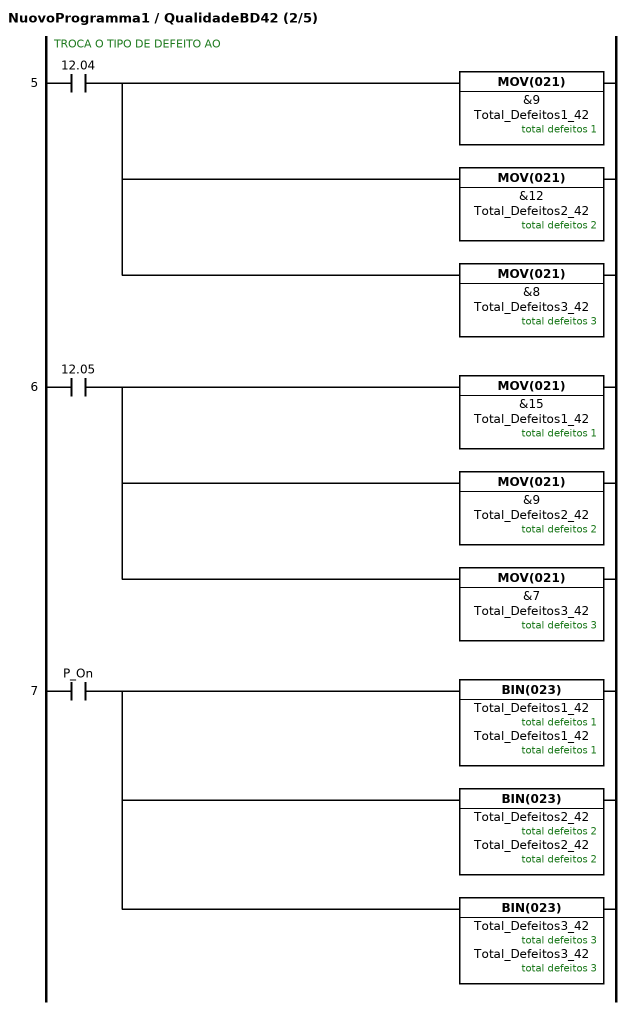
; [picture p24: NuovoProgramma1 / QualidadeBD42, rungs 5-7]
; rung 5: TROCA O TIPO DE DEFEITO AO
LD 12.04
MOV(021) &9 Total_Defeitos1_42  ; total defeitos 1
MOV(021) &12 Total_Defeitos2_42  ; total defeitos 2
MOV(021) &8 Total_Defeitos3_42  ; total defeitos 3
; rung 6
LD 12.05
MOV(021) &15 Total_Defeitos1_42  ; total defeitos 1
MOV(021) &9 Total_Defeitos2_42  ; total defeitos 2
MOV(021) &7 Total_Defeitos3_42  ; total defeitos 3
; rung 7
LD P_On
BIN(023) Total_Defeitos1_42 Total_Defeitos1_42  ; total defeitos 1
BIN(023) Total_Defeitos2_42 Total_Defeitos2_42  ; total defeitos 2
BIN(023) Total_Defeitos3_42 Total_Defeitos3_42  ; total defeitos 3

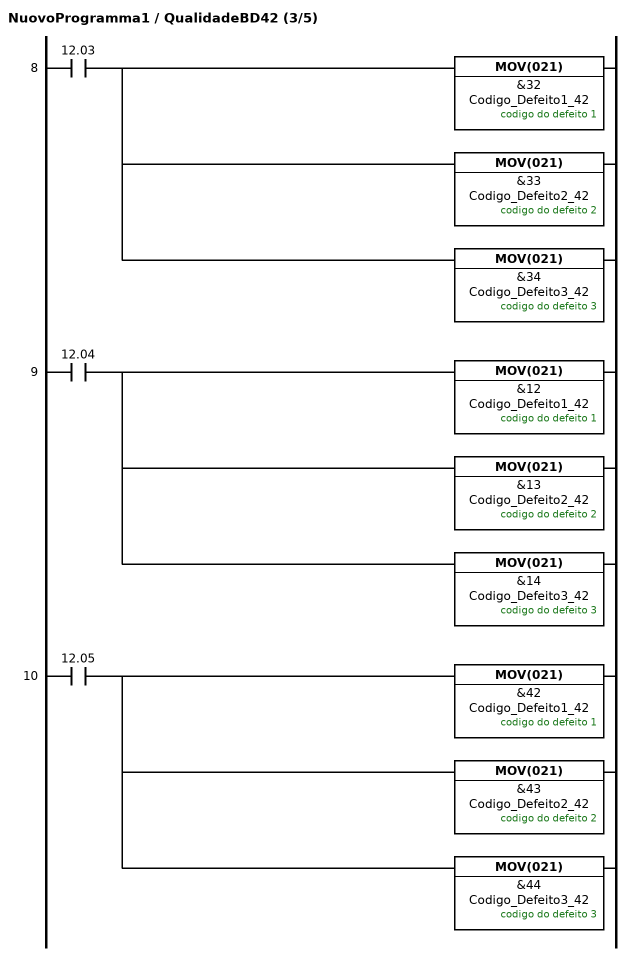
; rung 8
LD 12.03
MOV(021) &32 Codigo_Defeito1_42  ; codigo do defeito 1
MOV(021) &33 Codigo_Defeito2_42  ; codigo do defeito 2
MOV(021) &34 Codigo_Defeito3_42  ; codigo do defeito 3
; rung 9
LD 12.04
MOV(021) &12 Codigo_Defeito1_42  ; codigo do defeito 1
MOV(021) &13 Codigo_Defeito2_42  ; codigo do defeito 2
MOV(021) &14 Codigo_Defeito3_42  ; codigo do defeito 3
; rung 10
LD 12.05
MOV(021) &42 Codigo_Defeito1_42  ; codigo do defeito 1
MOV(021) &43 Codigo_Defeito2_42  ; codigo do defeito 2
MOV(021) &44 Codigo_Defeito3_42  ; codigo do defeito 3

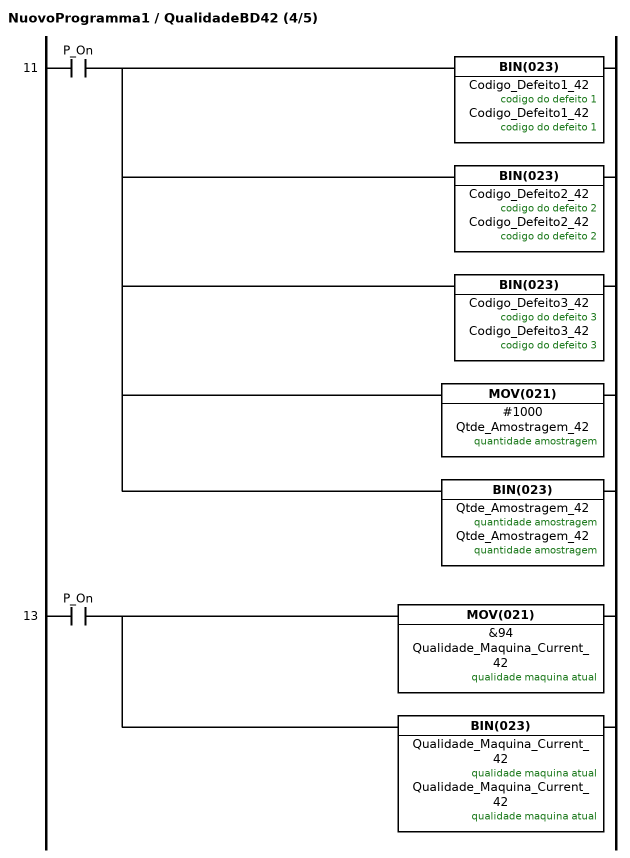
; rung 11
LD P_On
BIN(023) Codigo_Defeito1_42 Codigo_Defeito1_42  ; codigo do defeito 1
BIN(023) Codigo_Defeito2_42 Codigo_Defeito2_42  ; codigo do defeito 2
BIN(023) Codigo_Defeito3_42 Codigo_Defeito3_42  ; codigo do defeito 3
MOV(021) #1000 Qtde_Amostragem_42  ; quantidade amostragem
BIN(023) Qtde_Amostragem_42 Qtde_Amostragem_42  ; quantidade amostragem
; rung 13
LD P_On
MOV(021) &94 Qualidade_Maquina_Current_42  ; qualidade maquina atual
BIN(023) Qualidade_Maquina_Current_42 Qualidade_Maquina_Current_42  ; qualidade maquina atual

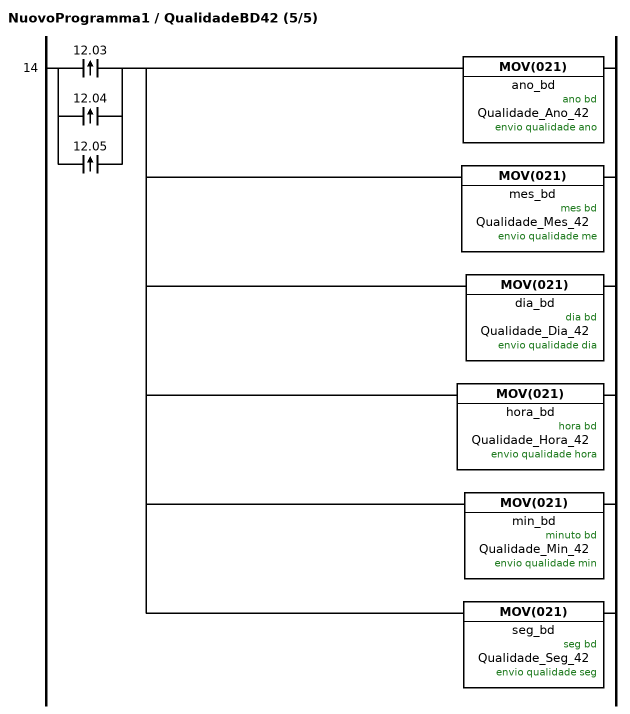
; rung 14
@LD 12.03
@OR 12.04
@OR 12.05
MOV(021) ano_bd Qualidade_Ano_42  ; ano bd, envio qualidade ano
MOV(021) mes_bd Qualidade_Mes_42  ; mes bd, envio qualidade me
MOV(021) dia_bd Qualidade_Dia_42  ; dia bd, envio qualidade dia
MOV(021) hora_bd Qualidade_Hora_42  ; hora bd, envio qualidade hora
MOV(021) min_bd Qualidade_Min_42  ; minuto bd, envio qualidade min
MOV(021) seg_bd Qualidade_Seg_42  ; seg bd, envio qualidade seg

### Section QualidadeBD43

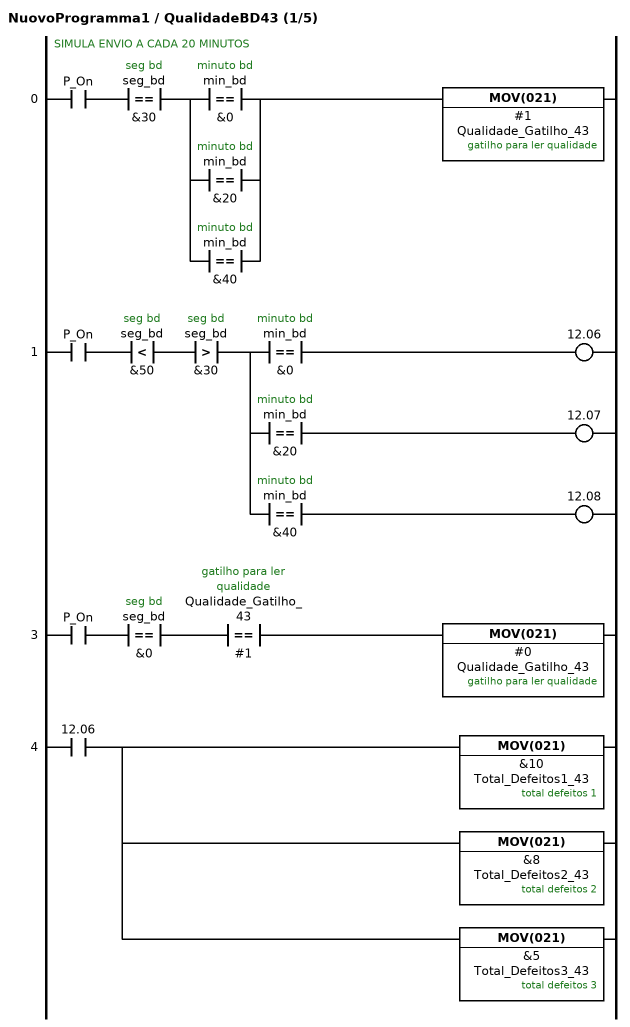
; rung 0: SIMULA ENVIO A CADA 20 MINUTOS
LD P_On
AND=(300) seg_bd &30  ; seg bd
LD=(300) min_bd &0  ; minuto bd
OR=(300) min_bd &20  ; minuto bd
OR=(300) min_bd &40  ; minuto bd
ANDLD
MOV(021) #1 Qualidade_Gatilho_43  ; gatilho para ler qualidade
; rung 1
LD P_On
AND<(310) seg_bd &50  ; seg bd
AND>(320) seg_bd &30  ; seg bd
OUT TR0
AND=(300) min_bd &0  ; minuto bd
OUT 12.06
LD TR0
AND=(300) min_bd &20  ; minuto bd
OUT 12.07
LD TR0
AND=(300) min_bd &40  ; minuto bd
OUT 12.08
; rung 3
LD P_On
AND=(300) seg_bd &0  ; seg bd
AND=(300) Qualidade_Gatilho_43 #1  ; gatilho para ler qualidade
MOV(021) #0 Qualidade_Gatilho_43  ; gatilho para ler qualidade
; rung 4
LD 12.06
MOV(021) &10 Total_Defeitos1_43  ; total defeitos 1
MOV(021) &8 Total_Defeitos2_43  ; total defeitos 2
MOV(021) &5 Total_Defeitos3_43  ; total defeitos 3

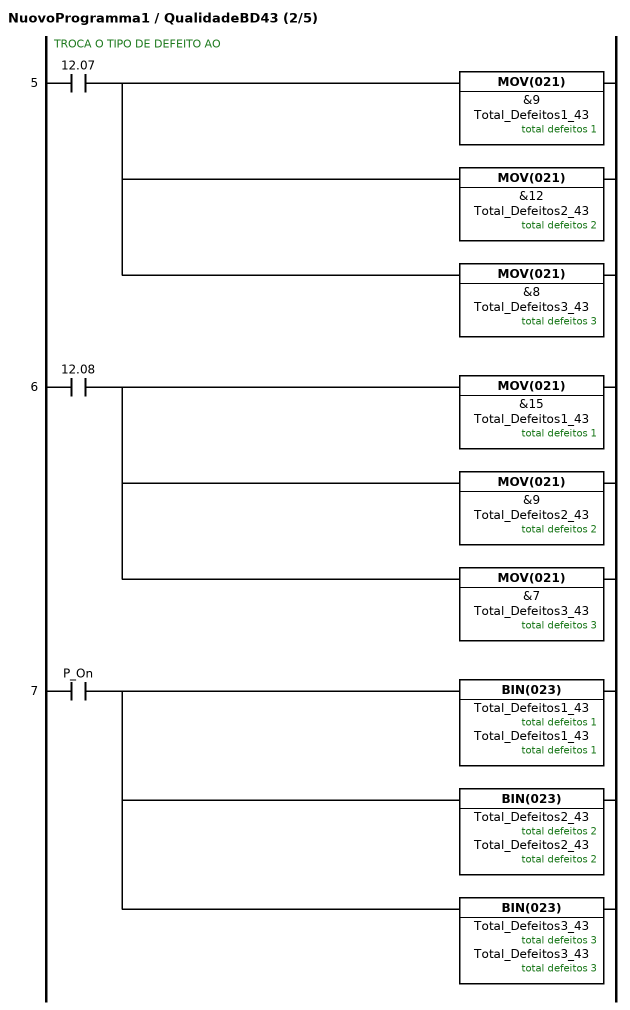
; rung 5: TROCA O TIPO DE DEFEITO AO
LD 12.07
MOV(021) &9 Total_Defeitos1_43  ; total defeitos 1
MOV(021) &12 Total_Defeitos2_43  ; total defeitos 2
MOV(021) &8 Total_Defeitos3_43  ; total defeitos 3
; rung 6
LD 12.08
MOV(021) &15 Total_Defeitos1_43  ; total defeitos 1
MOV(021) &9 Total_Defeitos2_43  ; total defeitos 2
MOV(021) &7 Total_Defeitos3_43  ; total defeitos 3
; rung 7
LD P_On
BIN(023) Total_Defeitos1_43 Total_Defeitos1_43  ; total defeitos 1
BIN(023) Total_Defeitos2_43 Total_Defeitos2_43  ; total defeitos 2
BIN(023) Total_Defeitos3_43 Total_Defeitos3_43  ; total defeitos 3

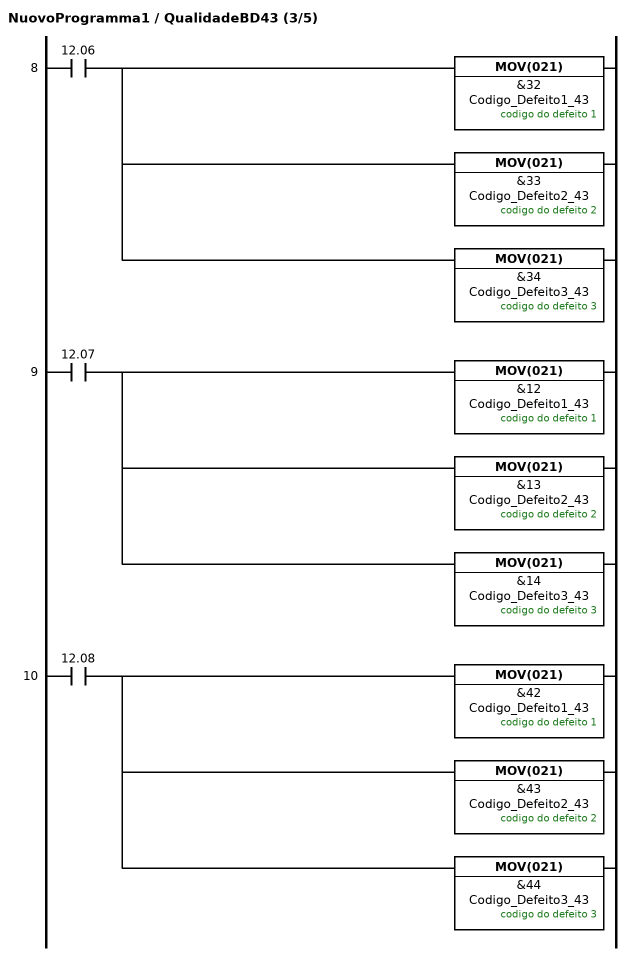
; rung 8
LD 12.06
MOV(021) &32 Codigo_Defeito1_43  ; codigo do defeito 1
MOV(021) &33 Codigo_Defeito2_43  ; codigo do defeito 2
MOV(021) &34 Codigo_Defeito3_43  ; codigo do defeito 3
; rung 9
LD 12.07
MOV(021) &12 Codigo_Defeito1_43  ; codigo do defeito 1
MOV(021) &13 Codigo_Defeito2_43  ; codigo do defeito 2
MOV(021) &14 Codigo_Defeito3_43  ; codigo do defeito 3
; rung 10
LD 12.08
MOV(021) &42 Codigo_Defeito1_43  ; codigo do defeito 1
MOV(021) &43 Codigo_Defeito2_43  ; codigo do defeito 2
MOV(021) &44 Codigo_Defeito3_43  ; codigo do defeito 3

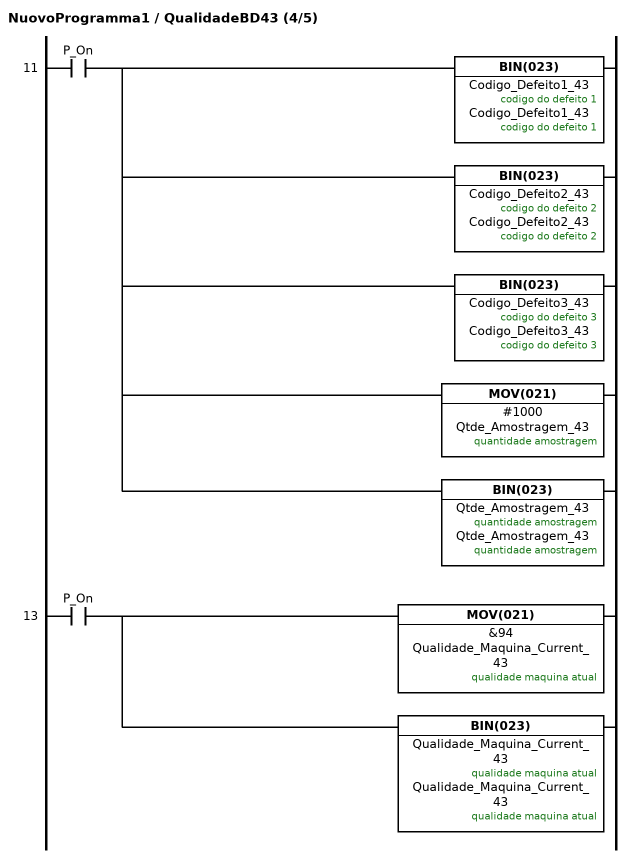
; rung 11
LD P_On
BIN(023) Codigo_Defeito1_43 Codigo_Defeito1_43  ; codigo do defeito 1
BIN(023) Codigo_Defeito2_43 Codigo_Defeito2_43  ; codigo do defeito 2
BIN(023) Codigo_Defeito3_43 Codigo_Defeito3_43  ; codigo do defeito 3
MOV(021) #1000 Qtde_Amostragem_43  ; quantidade amostragem
BIN(023) Qtde_Amostragem_43 Qtde_Amostragem_43  ; quantidade amostragem
; rung 13
LD P_On
MOV(021) &94 Qualidade_Maquina_Current_43  ; qualidade maquina atual
BIN(023) Qualidade_Maquina_Current_43 Qualidade_Maquina_Current_43  ; qualidade maquina atual

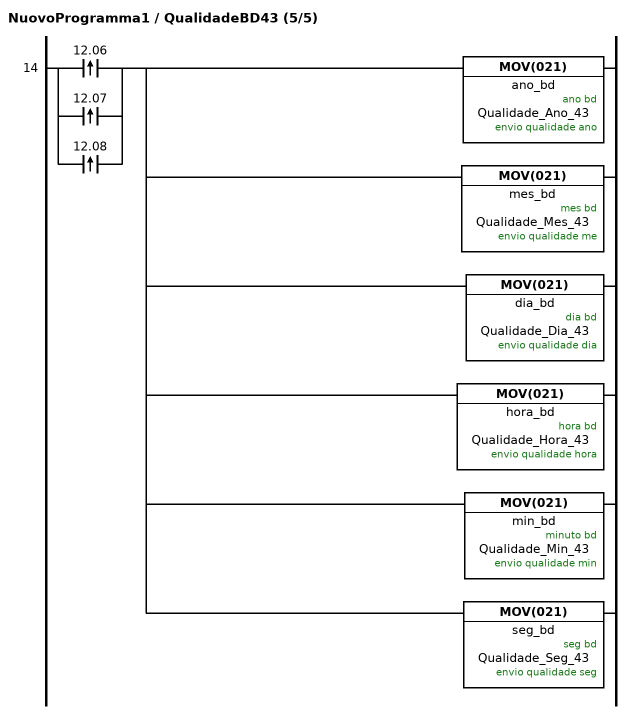
; rung 14
@LD 12.06
@OR 12.07
@OR 12.08
MOV(021) ano_bd Qualidade_Ano_43  ; ano bd, envio qualidade ano
MOV(021) mes_bd Qualidade_Mes_43  ; mes bd, envio qualidade me
MOV(021) dia_bd Qualidade_Dia_43  ; dia bd, envio qualidade dia
MOV(021) hora_bd Qualidade_Hora_43  ; hora bd, envio qualidade hora
MOV(021) min_bd Qualidade_Min_43  ; minuto bd, envio qualidade min
MOV(021) seg_bd Qualidade_Seg_43  ; seg bd, envio qualidade seg

### Section END
; rung 0
END(001)

## Function block Contador_de_Peças_PH29
VAR_INPUT
  Relógio_horas : WORD;
  Relógio_minutos : WORD;
  Dia_calendario : WORD;
  Mês_calendario : WORD;
  Contador : BOOL;
END_VAR
VAR
  _31dias_vezes_2 AT D520 : WORD;
  Ponteiro_DWord AT D522 : WORD;
  Memória_de_Armazenagem AT D524 : WORD;
  Memoria_contagem_BIN AT D526 : WORD;
  Memoria_contagem_BCD AT D528 : WORD;
END_VAR

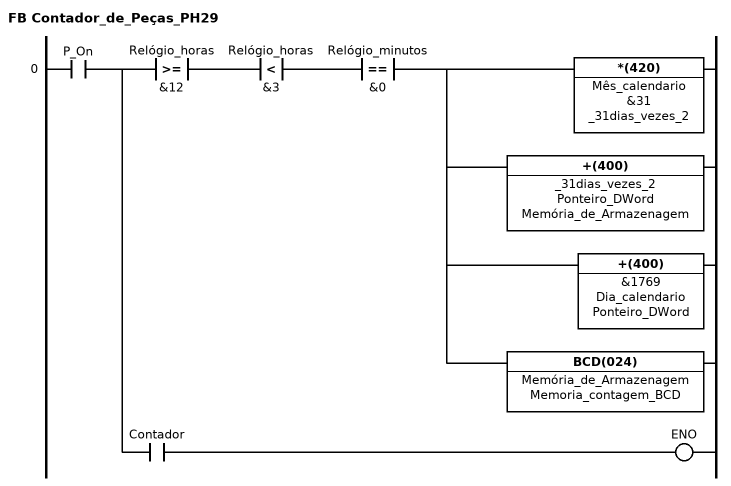
; rung 0
LD P_On
OUT TR0
AND>=(325) Relógio_horas &12
AND<(310) Relógio_horas &3
AND=(300) Relógio_minutos &0
*(420) Mês_calendario &31 _31dias_vezes_2
+(400) _31dias_vezes_2 Ponteiro_DWord Memória_de_Armazenagem
+(400) &1769 Dia_calendario Ponteiro_DWord
BCD(024) Memória_de_Armazenagem Memoria_contagem_BCD
LD TR0
AND Contador
OUT ENO

## Function block Contador_de_Peças_PH30
VAR_INPUT
  Relógio_horas : WORD;
  Relógio_minutos : WORD;
  Dia_calendario : WORD;
  Mês_calendario : WORD;
  Contador : BOOL;
END_VAR
VAR
  _31dias_vezes_2 AT D510 : WORD;
  Ponteiro_DWord AT D512 : WORD;
  Memória_de_Armazenagem AT D514 : WORD;
  Memoria_contagem_BIN AT D516 : WORD;
  Memoria_contagem_BCD AT D518 : WORD;
END_VAR

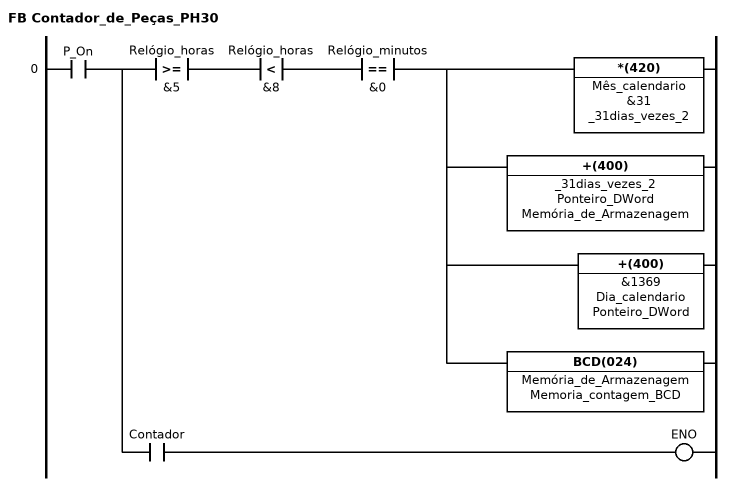
; rung 0
LD P_On
OUT TR0
AND>=(325) Relógio_horas &5
AND<(310) Relógio_horas &8
AND=(300) Relógio_minutos &0
*(420) Mês_calendario &31 _31dias_vezes_2
+(400) _31dias_vezes_2 Ponteiro_DWord Memória_de_Armazenagem
+(400) &1369 Dia_calendario Ponteiro_DWord
BCD(024) Memória_de_Armazenagem Memoria_contagem_BCD
LD TR0
AND Contador
OUT ENO

## Function block Contador_de_Peças_PH31
VAR_INPUT
  Relógio_horas : WORD;
  Relógio_minutos : WORD;
  Dia_calendario : WORD;
  Mês_calendario : WORD;
  Contador : BOOL;
END_VAR
VAR
  _31dias_vezes_2 AT D500 : WORD;
  Ponteiro_DWord AT D502 : WORD;
  Memória_de_Armazenagem AT D504 : WORD;
  Memoria_contagem_BIN AT D506 : WORD;
  Memoria_contagem_BCD AT D508 : WORD;
END_VAR

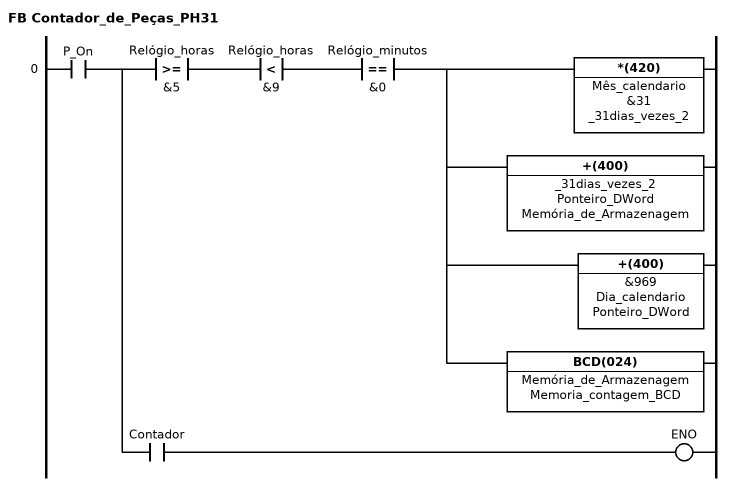
; rung 0
LD P_On
OUT TR0
AND>=(325) Relógio_horas &5
AND<(310) Relógio_horas &9
AND=(300) Relógio_minutos &0
*(420) Mês_calendario &31 _31dias_vezes_2
+(400) _31dias_vezes_2 Ponteiro_DWord Memória_de_Armazenagem
+(400) &969 Dia_calendario Ponteiro_DWord
BCD(024) Memória_de_Armazenagem Memoria_contagem_BCD
LD TR0
AND Contador
OUT ENO

## Function block Formato_de_Trabalho_29
VAR_INPUT
  Dia_calendario : WORD;
  Mês_calendario : WORD;
END_VAR
VAR
  _31dias_vezes_2 AT D546 : WORD;
  Ponteiro_DWord AT D548 : WORD;
  Memória_de_Armazenagem AT D550 : WORD;
  Memoria_contagem_BCD AT D552 : WORD;
END_VAR

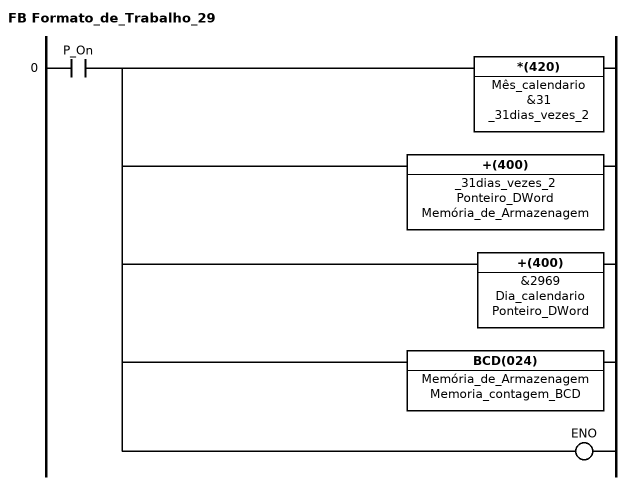
; rung 0
LD P_On
*(420) Mês_calendario &31 _31dias_vezes_2
+(400) _31dias_vezes_2 Ponteiro_DWord Memória_de_Armazenagem
+(400) &2969 Dia_calendario Ponteiro_DWord
BCD(024) Memória_de_Armazenagem Memoria_contagem_BCD
OUT ENO

## Function block Formato_de_Trabalho_30
VAR_INPUT
  Dia_calendario : WORD;
  Mês_calendario : WORD;
END_VAR
VAR
  _31dias_vezes_2 AT D538 : WORD;
  Ponteiro_DWord AT D540 : WORD;
  Memória_de_Armazenagem AT D542 : WORD;
  Memoria_contagem_BCD AT D544 : WORD;
END_VAR

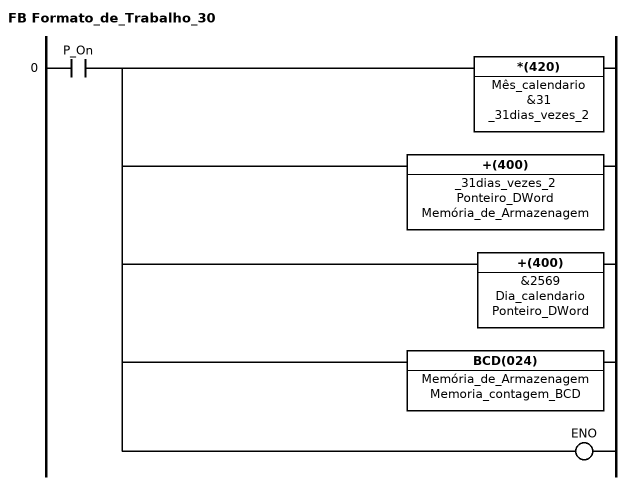
; rung 0
LD P_On
*(420) Mês_calendario &31 _31dias_vezes_2
+(400) _31dias_vezes_2 Ponteiro_DWord Memória_de_Armazenagem
+(400) &2569 Dia_calendario Ponteiro_DWord
BCD(024) Memória_de_Armazenagem Memoria_contagem_BCD
OUT ENO

## Function block Formato_de_Trabalho_31
VAR_INPUT
  Dia_calendario : WORD;
  Mês_calendario : WORD;
END_VAR
VAR
  _31dias_vezes_2 AT D530 : WORD;
  Ponteiro_DWord AT D532 : WORD;
  Memória_de_Armazenagem AT D534 : WORD;
  Memoria_contagem_BCD AT D536 : WORD;
END_VAR

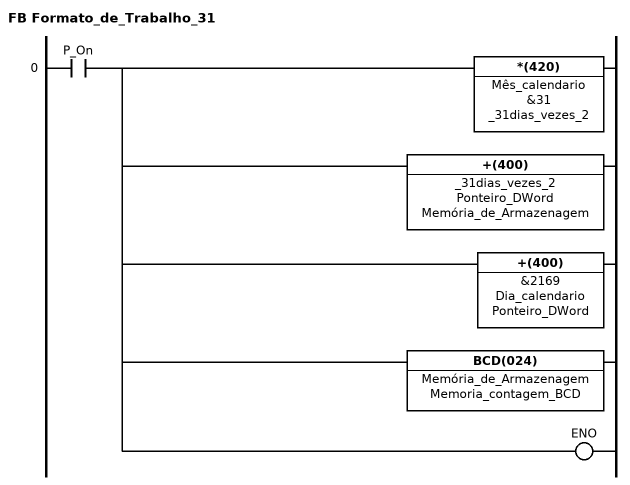
; rung 0
LD P_On
*(420) Mês_calendario &31 _31dias_vezes_2
+(400) _31dias_vezes_2 Ponteiro_DWord Memória_de_Armazenagem
+(400) &2169 Dia_calendario Ponteiro_DWord
BCD(024) Memória_de_Armazenagem Memoria_contagem_BCD
OUT ENO